PROGRAM MAIN
VAR
    machine1 : FB_SortingMachine;
    machine2 : FB_SortingMachine;
    machine3 : FB_SortingMachine;
END_VAR

machine1(machineID := 1);
machine2(machineID := 2);
machine3(machineID := 3);

END_PROGRAM

(* stored: Version 1.1.0.1
   POU MAIN: Id {67f882fd-9727-4250-b183-8627148893e5}, SpecialFunc None *)
